FUNCTION Convert_SINT_TO_STRING : Hresult
VAR_INPUT
	in : SINT;
	out : REFERENCE TO STRING;
END_VAR
VAR
	converted : STRING;
END_VAR
VAR CONSTANT
	INCOMPATIBLE : HRESULT := 16#9811070E;
END_VAR

converted := SINT_TO_STRING(in);

IF (STRING_TO_SINT(converted) <> in) THEN
	Convert_SINT_TO_STRING := INCOMPATIBLE;
	RETURN;
END_IF

out := converted;

END_FUNCTION

(* stored: Version 1.1.0.1, ProductVersion 3.1.4024.12
   POU Convert_SINT_TO_STRING: Id {6d9bec10-165b-468b-99a0-aa74b36ce0d4}, SpecialFunc None *)
